(*
SPDX-FileCopyrightText: © 2026 Oleksandr Tiutyk <trofimich@gmail.com>
SPDX-License-Identifier: MIT
License: https://opensource.org/license/mit
*)

{attribute 'qualified_only'}
{attribute 'strict'}
{attribute 'to_string'}
TYPE LOAD_STATE :
(
	NOT_LOADED,
	LOADING,
	LOADED,
	FAILED
);
END_TYPE

(* stored: Version 1.1.0.1
   DUT LOAD_STATE: Id {778d15df-dac5-43ec-99db-4178d3b4eae2} *)
